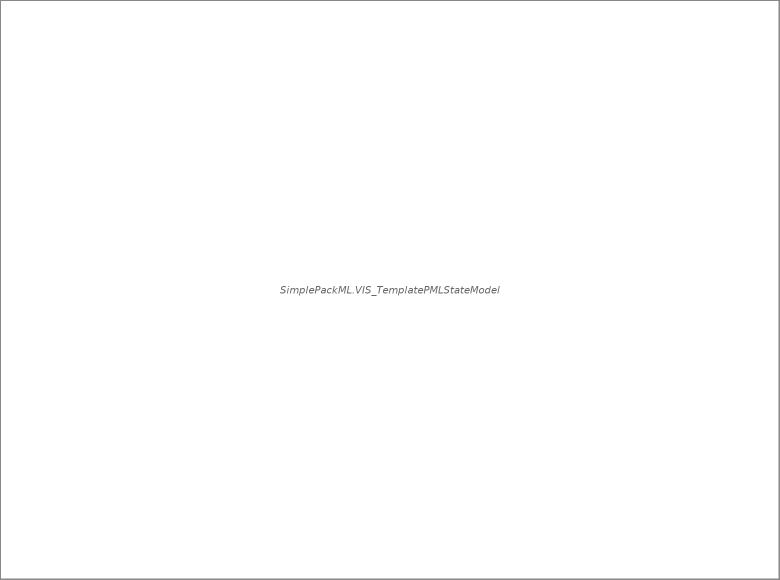
VISUALIZATION Visualization  // 780x580
    Frame (0,0 780x580)
        shows SimplePackML.VIS_TemplatePMLStateModel(ePMLUnitMode := P_PackML.machine1.eMode, ePMLState := P_PackML.machine1.eState)
END_VISUALIZATION

(* stored: Version 1.1.0.1
   Visu Visualization: Id {bce98e92-c157-41fe-a545-2ec1a48e0853} *)
